FUNCTION_BLOCK M1M2IO EXTENDS SM_M1M2IO
VAR_INPUT
END_VAR
VAR_OUTPUT
END_VAR
VAR
    _testVar_M1M2IO : BOOL;
END_VAR

SUPER^();

END_FUNCTION_BLOCK

(* stored: Version 1.1.0.1, ProductVersion 3.1.4018.2
   POU M1M2IO: Id {ccc8ad36-63ff-4126-9530-fea3e2775d63}, SpecialFunc None *)
